// TIA Portal project "LearningFactory_4_0_24V_Task06_MultiProcessingMPO" (V16)

(* hardware
DEVICE "ET 200SP-Station_1"  ET 200SP-Station
   slot 0: "Baugruppenträger_0"  Rack  6ES5 710-8MAx1
   slot 1: "PLC"  CPU 1512SP-1 PN  6ES7 512-1DK01-0AB0  V2.8
      slot 32768: "PROFINET"  X1
   slot 2: "DO1+2"  DQ 16x24VDC/0.5A ST  6ES7 132-6BH01-0BA0  V0.0
      slot 1: "DO1+2"  DQ 16x24VDC/0.5A ST
   slot 3: "DO3+4"  DQ 16x24VDC/0.5A ST  6ES7 132-6BH01-0BA0  V0.0
      slot 1: "DO3+4"  DQ 16x24VDC/0.5A ST
   slot 4: "DO5+6"  DQ 16x24VDC/0.5A ST  6ES7 132-6BH01-0BA0  V0.0
      slot 1: "DO5+6"  DQ 16x24VDC/0.5A ST
   slot 5: "DO7-14"  DQ 4x24VDC/2A HS  6ES7 132-6BD20-0DA0  V2.0
      slot 1: "DO7-14"  DQ 4x24VDC/2A HS
   slot 6: "DO15-22"  DQ 4x24VDC/2A HS  6ES7 132-6BD20-0DA0  V2.0
      slot 1: "DO15-22"  DQ 4x24VDC/2A HS
   slot 7: "DO23-30"  DQ 4x24VDC/2A HS  6ES7 132-6BD20-0DA0  V2.0
      slot 1: "DO23-30"  DQ 4x24VDC/2A HS
   slot 8: "DI1+2"  DI 16x24VDC ST  6ES7 131-6BH01-0BA0  V0.0
      slot 1: "DI1+2"  DI 16x24VDC ST
   slot 9: "DI3+4"  DI 16x24VDC ST  6ES7 131-6BH01-0BA0  V0.0
      slot 1: "DI3+4"  DI 16x24VDC ST
   slot 10: "DI5"  DI 8x24VDC HS  6ES7 131-6BF00-0DA0  V1.0
      slot 1: "DI5"  DI 8x24VDC HS
   slot 11: "DI6"  DI 8x24VDC HS  6ES7 131-6BF00-0DA0  V1.0
      slot 1: "DI6"  DI 8x24VDC HS
   slot 12: "AI7-10"  AI 2xU ST  6ES7 134-6FB00-0BA1  V1.0
      slot 1: "AI7-10"  AI 2xU ST
   slot 13: "End"  Server module  6ES7 193-6PA00-0AA0  V1.1
      slot 1: "End"  Server module
   slot 127: "BA 2xRJ45"  BA 2xRJ45  6ES7 193-6AR00-0AA0  V0.0
      slot 32769: "Port_1"  6ES7 193-6AR00-0AA0
      slot 32770: "Port_2"  6ES7 193-6AR00-0AA0
*)

// ===== PLC "PLC"  CPU 1512SP-1 PN =====

VAR_GLOBAL   // PLC tag table "Start_Stop"
   "IX_START" AT %I4.4 : Bool;
   "IX_STOP" AT %I4.6 : Bool;
END_VAR

VAR_GLOBAL   // PLC tag table "MPO - Multi Processing Station with Oven"
   "IX_MPO_RefSwitchTurnTable_PosVac_I1" AT %I1.7 : Bool;
   "IX_MPO_RefSwitchTurnTable_PosBelt_I2" AT %I2.0 : Bool;
   "IX_MPO_LightBarrierEndOfConBelt_I3" AT %I2.1 : Bool;
   "IX_MPO_RefSwitchTurnTable_PosSaw_I4" AT %I2.2 : Bool;
   "IX_MPO_RefSwitchVac_PosTurnTable_I5" AT %I2.3 : Bool;
   "IX_MPO_RefSwitchOvenFeederInside_I6" AT %I2.4 : Bool;
   "IX_MPO_RefSwitchOvenFeederOutside_I7" AT %I2.5 : Bool;
   "IX_MPO_RefSwitchVac_PosOven_I8" AT %I2.6 : Bool;
   "IX_MPO_LightBarrierOven_I9" AT %I2.7 : Bool;
   "QX_MPO_M1_TurnTableClockwise_Q1" AT %Q3.0 : Bool;
   "QX_MPO_M1_TurnTableCounterclockwise_Q2" AT %Q3.1 : Bool;
   "QX_MPO_M2_ConveyorBeltForward_Q3" AT %Q3.2 : Bool;
   "QX_MPO_M3_Saw_Q4" AT %Q3.3 : Bool;
   "QX_MPO_M4_OvenFeederRetract_Q5" AT %Q3.4 : Bool;
   "QX_MPO_M4_OvenFeederExtend_Q6" AT %Q3.5 : Bool;
   "QX_MPO_M5_VacuumTowardsOven_Q7" AT %Q3.6 : Bool;
   "QX_MPO_M5_VacuumTowardsTurnTable_Q8" AT %Q3.7 : Bool;
   "QX_MPO_LightOven_Q9" AT %Q4.0 : Bool;
   "QX_MPO_Compressor_Q10" AT %Q4.1 : Bool;
   "QX_MPO_ValveVacuum_Q11" AT %Q4.2 : Bool;
   "QX_MPO_ValveLowering_Q12" AT %Q4.3 : Bool;
   "QX_MPO_ValveOvenDoor_Q13" AT %Q4.4 : Bool;
   "QX_MPO_ValveFeeder_Q14" AT %Q4.5 : Bool;
   "QW_MPO_PWM_TurnTable_M1" AT %QW23 : Int;
   "QW_MPO_PWM_Vacuum_M5" AT %QW25 : Int;
END_VAR

DATA_BLOCK "Task06_MultiProcessing_DB"   // DB4
{ S7_Optimized_Access := 'TRUE' }
VERSION : 0.1
// stored: InstanceOfName Task06_MultiProcessing
"Task06_MultiProcessing"
BEGIN
END_DATA_BLOCK

FUNCTION_BLOCK "Task06_MultiProcessing"   // FB4, SCL
{ S7_Optimized_Access := 'TRUE' }
VERSION : 0.1
   VAR_INPUT
      Start : Bool;
      Stop : Bool;
      RefSwitchTurnTable_PosVac : Bool;
      RefSwitchTurnTable_PosBelt : Bool;
      RefSwitchTurnTable_PosSaw : Bool;
      RefSwitchVac_PosTurnTable : Bool;
      RefSwitchVac_PosOven : Bool;
      RefSwitchOvenFeederInside : Bool;
      RefSwitchOvenFeederOutside : Bool;
      LightBarrierOven : Bool;
      LightBarrierEndOfConBelt : Bool;
   END_VAR
   VAR_OUTPUT
      M2_ConveyorBeltForward : Bool;
      M3_Saw : Bool;
      M4_OvenFeederRetract : Bool;
      M4_OvenFeederExtend : Bool;
      LightOven : Bool;
      PWM_TurnTable : Int;
      PWM_Vacuum : Int;
      Compressor : Bool;
   END_VAR
   VAR_IN_OUT
      M1_TurnTableClockwise : Bool;
      M1_TurnTableCounterclockwise : Bool;
      M5_VacuumTowardsOven : Bool;
      M5_VacuumTowardsTurnTable : Bool;
      ValveVacuum : Bool;
      ValveLowering : Bool;
      ValveOvenDoor : Bool;
      ValveFeeder : Bool;
   END_VAR
   VAR
      Step_number : Int;
      IEC_Timer_LoweringDown : TON_TIME;
      IEC_Timer_VacuumOn : TON_TIME;
      IEC_Timer_LoweringUp : TON_TIME;
      IEC_Timer_VacuumOff : TON_TIME;
      IEC_Timer_OvenClose : TON_TIME;
      IEC_Timer_OvenLight : TON_TIME;
      IEC_Timer_OvenOpen : TON_TIME;
      IEC_Timer_Saw : TON_TIME;
   END_VAR
BEGIN


   // Reset sequencer with pushbutton STOP 
   // Rücksetzen der Schrittkette  mit Taster STOP

   IF #Stop THEN
       #Step_number := 0;
   END_IF;

   // Start sequencer with pushbutton START
   // Starten der Schrittkette  mit Taster START

   CASE #Step_number OF
       0:  // Initial step 1 / Initialschritt 1
           #M2_ConveyorBeltForward := FALSE;           // Conveyor stop / Band stoppen  
           #M3_Saw := FALSE;                           // Saw off / Säge aus
           #M4_OvenFeederRetract := FALSE;             // Feeder oven retract stop / Ausschub Ofen einfahren stoppen
           #M4_OvenFeederExtend := FALSE;              // Feeder oven extend stop / Ausschub Ofen ausfahren stoppen 
           #LightOven := FALSE;                        // Light oven off / Licht im Ofen aus
           #M1_TurnTableClockwise := FALSE;            // Rotation clockwise stop / Rotation im Uhrzeigersinn stoppen
           #M1_TurnTableCounterclockwise := FALSE;     // Rotation counter clockwise stop / Rotation gegen den Uhrzeigersinn stoppen
           #M5_VacuumTowardsOven := FALSE;             // Linear axle towards oven stop / Linearachse zum Ofen stop 
           #M5_VacuumTowardsTurnTable := FALSE;        // Linear axle towards turn-table stop / Linearachse zum Drehtisch stop 
           #ValveVacuum := FALSE;                      // Vacuum gripper off / Vakuumgreifer aus
           #ValveLowering := FALSE;                    // Vacuum gripper up / Vakuumgreifer hoch
           #ValveOvenDoor := FALSE;                    // Door Oven close / Ofentüre schließen
           #ValveFeeder := FALSE;                      // Retract Zylinder feeder / Ausschubzylinder einfahren
           RESET_TIMER(#IEC_Timer_LoweringDown);       // Reset timer vacuum gripper down / Rücksetzen des Timers Vakuumgreifer abwärts
           RESET_TIMER(#IEC_Timer_VacuumOn);           // Reset timer vacuum on / Rücksetzen des Timers Vakuum ein
           RESET_TIMER(#IEC_Timer_LoweringUp);         // Reset timer vacuum gripper up / Rücksetzen des Timers Vakuumgreifer aufwärts
           RESET_TIMER(#IEC_Timer_VacuumOff);          // Reset timer vacuum off / Rücksetzen des Timers Vakuum aus
           RESET_TIMER(#IEC_Timer_OvenClose);          // Reset timer oven close / Rücksetzen des Timers Ofen schließen
           RESET_TIMER(#IEC_Timer_OvenLight);          // Reset timer light oven / Rücksetzen des Timers Licht im Ofen
           RESET_TIMER(#IEC_Timer_OvenOpen);           // Reset timer oven open / Rücksetzen des Timers Ofen öffnen
           RESET_TIMER(#IEC_Timer_Saw);                // Reset timer saw / Rücksetzen des Timers Säge

           IF #Start THEN
               #Step_number := #Step_number + 1;
           END_IF;

       1:  // Step 1 open oven; turn-table to position vacuum; linear axle towards turn-table
           // Schritt 1 Ofen öffnen; Drehtisch zu Position Vakuum; Linearachse zu Position Drehtisch
           #ValveOvenDoor := TRUE;                     // Door Oven open / Ofentüre öffnen
           #M1_TurnTableCounterclockwise := TRUE;      // Rotation counter clockwise / Rotation gegen den Uhrzeigersinn
           #M5_VacuumTowardsTurnTable := TRUE;         //Linear axle towards turn-table / Linearachse zum Drehtisch 

           IF #RefSwitchTurnTable_PosVac THEN
               #M1_TurnTableCounterclockwise := FALSE; // Rotation counter clockwise stop / Rotation gegen den Uhrzeigersinn stoppen
           END_IF;
           IF #RefSwitchVac_PosTurnTable THEN
               #M5_VacuumTowardsTurnTable := FALSE;    //Linear axle towards turn-table stop / Linearachse zum Drehtisch stop
           END_IF;

           IF #RefSwitchTurnTable_PosVac AND #RefSwitchVac_PosTurnTable THEN
               #Step_number := #Step_number + 1;
           END_IF;

       2:  // Step 2 vacuum gripper down / Schritt 2 Vakuumgreifer abwärts
           #ValveLowering := TRUE;                         // Vacuum gripper down / Vakuumgreifer abwärts
           #IEC_Timer_LoweringDown(IN := #ValveLowering,  // Start Timer vacuum gripper down / Timer starten Vakuumgreifer abwärts
                                PT := T#1s);

            IF #IEC_Timer_LoweringDown.Q THEN
                #Step_number := #Step_number + 1;
            END_IF;

        3:  // Step 3 vacuum on / Schritt 3 Vakuum ein
            #ValveVacuum := TRUE;                          // Vacuum on / Vakuum ein
            RESET_TIMER(#IEC_Timer_LoweringDown);          // Reset timer vacuum gripper down / Rücksetzen des Timers Vakuumgreifer abwärts
            #IEC_Timer_VacuumOn(IN := #ValveVacuum,        // Start Timer vacuum on / Timer starten Vakuum ein
                                    PT := T#1s);

            IF #IEC_Timer_VacuumOn.Q THEN
                #Step_number := #Step_number + 1;
            END_IF;

        4:  // Step 4 vacuum gripper up / Schritt 4 Vakuumgreifer aufwärts
            #ValveLowering := FALSE;                           // Vacuum gripper up / Vakuumgreifer aaufwärts
            RESET_TIMER(#IEC_Timer_VacuumOn);                  // Reset timer vacuum on / Rücksetzen des Timers Vakuum ein
            #IEC_Timer_LoweringUp(IN := NOT #ValveLowering,    // Start Timer vacuum gripper up / Timer starten Vakuumgreifer aufwärts
                                    PT := T#2s);

              IF #IEC_Timer_LoweringUp.Q THEN
                #Step_number := #Step_number + 1;
            END_IF;

        5:  // Step 5 extend feeder oven; linear axle towards oven
            // Schritt 5 Ausschub Ofen ausfahren; Linearachse zu Position Ofen
            #M4_OvenFeederExtend := TRUE;              // Feeder oven extend / Ausschub Ofen ausfahren 
            #M5_VacuumTowardsOven := TRUE;             // Linear axle towards oven / Linearachse zum Ofen
            RESET_TIMER(#IEC_Timer_LoweringUp);         // Reset timer vacuum gripper up / Rücksetzen des Timers Vakuumgreifer aufwärts

            IF #RefSwitchOvenFeederOutside THEN
                #M4_OvenFeederExtend := FALSE;         // Feeder oven extend stop / Ausschub Ofen ausfahren stoppen
            END_IF;
            IF #RefSwitchVac_PosOven THEN
                #M5_VacuumTowardsOven := FALSE;        //Linear axle towards oven stop / Linearachse zum Ofen stoppen
            END_IF;

            IF #RefSwitchOvenFeederOutside AND #RefSwitchVac_PosOven AND NOT #LightBarrierOven THEN
                #Step_number := #Step_number + 1;
            END_IF;

        6:  // Step 6 vacuum gripper down / Schritt 6 Vakuumgreifer abwärts
            #ValveLowering := TRUE;                         // Vacuum gripper down / Vakuumgreifer abwärts
            #IEC_Timer_LoweringDown(IN := #ValveLowering,  // Start Timer vacuum gripper down / Timer starten Vakuumgreifer abwärts
                                    PT := T#1s);

            IF #IEC_Timer_LoweringDown.Q THEN
                #Step_number := #Step_number + 1;
            END_IF;

        7:  // Step 7 vacuum off / Schritt 7 Vakuum aus
            #ValveVacuum := FALSE;                         // Vacuum off / Vakuum aus
            RESET_TIMER(#IEC_Timer_LoweringDown);          // Reset timer vacuum gripper down / Rücksetzen des Timers Vakuumgreifer abwärts
            #IEC_Timer_VacuumOff (IN := NOT #ValveVacuum,  // Start Timer vacuum off / Timer starten Vakuum off
                                PT := T#1s);

              IF #IEC_Timer_VacuumOff.Q THEN
                  #Step_number := #Step_number + 1;
              END_IF;

        8:  // Step 8 vacuum gripper up / Schritt 8 Vakuumgreifer aufwärts
            #ValveLowering := FALSE;                           // Vacuum gripper up / Vakuumgreifer aaufwärts
            RESET_TIMER(#IEC_Timer_VacuumOff);                 // Reset timer vacuum off / Rücksetzen des Timers Vakuum aus
            #IEC_Timer_LoweringUp(IN := NOT #ValveLowering,    // Start Timer vacuum gripper up / Timer starten Vakuumgreifer aufwärts
                                  PT := T#1s);

            IF #IEC_Timer_LoweringUp.Q THEN
                #Step_number := #Step_number + 1;
            END_IF;

        9:  // Step 9 retract feeder oven / Schritt 9 Ausschub Ofen einfahren
            #M4_OvenFeederRetract := TRUE;              // Feeder oven retract / Ausschub Ofen einfahren 
            RESET_TIMER(#IEC_Timer_LoweringUp);         // Reset Timer vacuum gripper up / Rücksetzen des Timers Vakuumgreifer aufwärts

            IF #RefSwitchOvenFeederInside THEN
                #Step_number := #Step_number + 1;
            END_IF;

       10:  // Step 10 close oven / Schritt 10 Ofen schließen
            #M4_OvenFeederRetract := FALSE;                    // Feeder oven retract off / Ausschub Ofen einfahren aus
            #ValveOvenDoor := FALSE;                           // Door Oven close / Ofentüre schließen
           #IEC_Timer_OvenClose(IN := NOT #ValveOvenDoor,     // Start Timer oven close / Starten des Timers Ofen schließen
                                  PT := T#1s);

             IF #IEC_Timer_OvenClose.Q THEN
                #Step_number := #Step_number + 1;
            END_IF;

        11:  // Step 11 light oven on / Schritt 11 Licht Ofen an
            #LightOven := TRUE;                        // Light oven on / Licht im Ofen an
            RESET_TIMER(#IEC_Timer_OvenClose);          // Reset timer oven close / Rücksetzen des Timers Ofen schließen
            #IEC_Timer_OvenLight(IN := #LightOven,     // Start Timer oven light / Starten des Timers Licht Ofen
                                 PT := T#5s);

            IF #IEC_Timer_OvenLight.Q THEN
                #Step_number := #Step_number + 1;
            END_IF;

        12:  // Step 12 open oven / Schritt 12 Ofen öffnen
            #LightOven := FALSE;                           // Light oven off / Licht im Ofen aus
            #ValveOvenDoor := TRUE;                        // Door Oven open / Ofentüre öffnen
            RESET_TIMER(#IEC_Timer_OvenLight);             // Reset timer light oven / Rücksetzen des Timers Licht im Ofen
            #IEC_Timer_OvenOpen(IN := #ValveOvenDoor,     // Start Timer oven open / Starten des Timers Ofen öffnen
                                 PT := T#1s);

             IF #IEC_Timer_OvenOpen.Q THEN
                #Step_number := #Step_number + 1;
            END_IF;

       13:  // Step 13 extend feeder oven / Schritt 13 Ausschub Ofen ausfahren
            #M4_OvenFeederExtend := TRUE;              // Feeder oven extend / Ausschub Ofen ausfahren 
            RESET_TIMER(#IEC_Timer_OvenOpen);           // Reset timer oven open / Rücksetzen des Timers Ofen öffnen

            IF #RefSwitchOvenFeederOutside THEN
                #Step_number := #Step_number + 1;
            END_IF;

       14:  // Step 14 vacuum gripper down; oven close / Schritt 14 Vakuumgreifer abwärts; Ofentüre schließen
            #ValveOvenDoor := FALSE;                        // Door Oven close / Ofentüre schließen
            #M4_OvenFeederExtend := FALSE;                  // Feeder oven extend off / Ausschub Ofen ausfahren aus
            #ValveLowering := TRUE;                         // Vacuum gripper down / Vakuumgreifer abwärts
            #IEC_Timer_LoweringDown(IN := #ValveLowering,  // Start Timer vacuum gripper down / Timer starten Vakuumgreifer abwärts
                                    PT := T#1s);

            IF #IEC_Timer_LoweringDown.Q THEN
                #Step_number := #Step_number + 1;
            END_IF;

       15:  // Step 15 vacuum on / Schritt 15 Vakuum ein
            #ValveVacuum := TRUE;                          // Vacuum on / Vakuum ein
            RESET_TIMER(#IEC_Timer_LoweringDown);          // Reset timer vacuum gripper down / Rücksetzen des Timers Vakuumgreifer abwärts
            #IEC_Timer_VacuumOn(IN := #ValveVacuum,        // Start Timer vacuum on / Timer starten Vakuum ein
                                PT := T#1s);

            IF #IEC_Timer_VacuumOn.Q THEN
                #Step_number := #Step_number + 1;
            END_IF;

        16:  // Step 16 vacuum gripper up / Schritt 16 Vakuumgreifer aufwärts
            #ValveLowering := FALSE;                           // Vacuum gripper up / Vakuumgreifer aaufwärts
            RESET_TIMER(#IEC_Timer_VacuumOn);                  // Reset timer vacuum on / Rücksetzen des Timers Vakuum ein
            #IEC_Timer_LoweringUp(IN := NOT #ValveLowering,    // Start Timer vacuum gripper up / Timer starten Vakuumgreifer aufwärts
                                  PT := T#2s);

            IF #IEC_Timer_LoweringUp.Q THEN
                #Step_number := #Step_number + 1;
            END_IF;

        17:  // Step 17 linear axle towards turn-table / Schritt 17 Linearachse zum Rundtisch
            #M5_VacuumTowardsTurnTable := TRUE;             // Linear axle towards turn-table / Linearachse zum Rundtisch
            RESET_TIMER(#IEC_Timer_LoweringUp);         // Reset timer vacuum gripper up / Rücksetzen des Timers Vakuumgreifer aufwärts

            IF #RefSwitchVac_PosTurnTable THEN
                #Step_number := #Step_number + 1;
            END_IF;

        18:  // Step 18 vacuum gripper down / Schritt 18 Vakuumgreifer abwärts
            #M5_VacuumTowardsTurnTable := FALSE;             // Linear axle towards turn-table off / Linearachse zum Rundtisch aus
            #ValveLowering := TRUE;                         // Vacuum gripper down / Vakuumgreifer abwärts
            #IEC_Timer_LoweringDown(IN := #ValveLowering,  // Start Timer vacuum gripper down / Timer starten Vakuumgreifer abwärts
                                    PT := T#1s);

            IF #IEC_Timer_LoweringDown.Q THEN
                #Step_number := #Step_number + 1;
            END_IF;

       19:  // Step 7 vacuum off / Schritt 19 Vakuum aus
            #ValveVacuum := FALSE;                         // Vacuum off / Vakuum aus
            RESET_TIMER(#IEC_Timer_LoweringDown);          // Reset timer vacuum gripper down / Rücksetzen des Timers Vakuumgreifer abwärts
            #IEC_Timer_VacuumOff(IN := NOT #ValveVacuum,  // Start Timer vacuum off / Timer starten Vakuum off
                                 PT := T#1s);

            IF #IEC_Timer_VacuumOff.Q THEN
                #Step_number := #Step_number + 1;
            END_IF;

       20:  // Step 20 vacuum gripper up / Schritt 20 Vakuumgreifer aufwärts
            #ValveLowering := FALSE;                           // Vacuum gripper up / Vakuumgreifer aaufwärts
            RESET_TIMER(#IEC_Timer_VacuumOff);                 // Reset timer vacuum off / Rücksetzen des Timers Vakuum aus
            #IEC_Timer_LoweringUp(IN := NOT #ValveLowering,    // Start Timer vacuum gripper up / Timer starten Vakuumgreifer aufwärts
                                  PT := T#1s);

            IF #IEC_Timer_LoweringUp.Q THEN
                #Step_number := #Step_number + 1;
            END_IF;

       21:  // Step 21 rotation clockwise to position saw / Schritt 21 Rotation im Uhrzeigersinn zur Position Säge
           #M1_TurnTableClockwise := TRUE;            // Rotation clockwise / Rotation im Uhrzeigersinn
            RESET_TIMER(#IEC_Timer_LoweringUp);         // Reset Timer vacuum gripper up / Rücksetzen des Timers Vakuumgreifer aufwärts

            IF #RefSwitchTurnTable_PosSaw THEN
                #Step_number := #Step_number + 1;
            END_IF;

       22:  // Step 22 saw on 5 seconds / Schritt 22 Säge ein 5 Sekunden
            #M1_TurnTableClockwise := FALSE;            // Rotation clockwise stop/ Rotation im Uhrzeigersinn stoppen
            #M3_Saw := TRUE;                           // Saw on / Säge ein
            #IEC_Timer_Saw(IN := #M3_Saw,    // Start Timer saw on / Timer starten Säge ein
                                  PT := T#5s);

            IF #IEC_Timer_Saw.Q THEN
                #Step_number := #Step_number + 1;
            END_IF;

       23:  // Step 23 rotation clockwise to position conveyorbelt/ Schritt 23 Rotation im Uhrzeigersinn zum Förderband
            #M3_Saw := FALSE;                           // Saw off / Säge aus
            #M1_TurnTableClockwise := TRUE;            // Rotation clockwise / Rotation im Uhrzeigersinn
            RESET_TIMER(#IEC_Timer_Saw);                // Reset timer saw / Rücksetzen des Timers Säge

            IF #RefSwitchTurnTable_PosBelt THEN
               #Step_number := #Step_number + 1;
           END_IF;

       24:  // Step 24 extend feeder; start conveyorbelt/ Schritt 24 Ausschubzylinder ausfahren; Band starten
               #M1_TurnTableClockwise := FALSE;            // Rotation clockwise off / Rotation im Uhrzeigersinn aus
               #ValveFeeder := TRUE;                      // Extend Zylinder feeder / Ausschubzylinder ausfahren
               #M2_ConveyorBeltForward := TRUE;           // Conveyorbelt start / Band starten 

               IF #LightBarrierEndOfConBelt THEN
                   #Step_number := #Step_number + 1;
               END_IF;

       25:  // Step 25 end of sequencer / Schritt 24 Schrittkettenende
               #ValveFeeder := FALSE;                          // Retract Zylinder feeder / Ausschubzylinder einfahren
               #M2_ConveyorBeltForward := FALSE;              // Conveyorbelt stop / Band stoppen

               IF NOT #ValveFeeder AND NOT #M2_ConveyorBeltForward THEN
                   #Step_number :=0;
               END_IF;

           ELSE  // Statement section ELSE
           ;
   END_CASE;


   //Permanent Instructions

   //Pulse width modulation control for turn-table 
   //Pulsweitenmodulation für Drehtisch
   IF #M1_TurnTableClockwise OR #M1_TurnTableCounterclockwise
   THEN
       #PWM_TurnTable := 500;
   ELSE
       #PWM_TurnTable := 0;
   END_IF;

   //Pulse width modulation control for linear axle vacuum gripper
   //Pulsweitenmodulation für Linearachse Vakuumgreifer
   IF #M5_VacuumTowardsOven OR #M5_VacuumTowardsTurnTable
   THEN
       #PWM_Vacuum := 700;
   ELSE
       #PWM_Vacuum := 0;
   END_IF;

   // Compressor on / Kompressor ein
   IF #ValveVacuum OR #ValveLowering
       OR #ValveOvenDoor OR #ValveFeeder
   THEN
       #Compressor := TRUE;
   ELSE
       #Compressor := FALSE;
   END_IF;
END_FUNCTION_BLOCK

ORGANIZATION_BLOCK "Main"   // OB1, SCL, ProgramCycle
TITLE = "Main Program Sweep (Cycle)"
{ S7_Optimized_Access := 'TRUE' }
VERSION : 0.1
   VAR_INPUT
      Initial_Call : Bool;   // Initial call of this OB
      Remanence : Bool;   // =True, if remanent data are available
   END_VAR
BEGIN


   // Call subroutine VacuumGripper
   // Aufruf Unterprogramm VacuumGripper


   "Task06_MultiProcessing_DB"(Start:="IX_START",
                               Stop:= NOT "IX_STOP",
                               RefSwitchTurnTable_PosVac:="IX_MPO_RefSwitchTurnTable_PosVac_I1",
                               RefSwitchTurnTable_PosBelt:="IX_MPO_RefSwitchTurnTable_PosBelt_I2",
                               RefSwitchTurnTable_PosSaw:="IX_MPO_RefSwitchTurnTable_PosSaw_I4",
                               RefSwitchVac_PosTurnTable:="IX_MPO_RefSwitchVac_PosTurnTable_I5",
                               RefSwitchVac_PosOven:="IX_MPO_RefSwitchVac_PosOven_I8",
                               RefSwitchOvenFeederInside:="IX_MPO_RefSwitchOvenFeederInside_I6",
                               RefSwitchOvenFeederOutside:="IX_MPO_RefSwitchOvenFeederOutside_I7",
                               LightBarrierOven:= NOT "IX_MPO_LightBarrierOven_I9",
                               LightBarrierEndOfConBelt:= NOT "IX_MPO_LightBarrierEndOfConBelt_I3",
                               M1_TurnTableClockwise:="QX_MPO_M1_TurnTableClockwise_Q1",
                               M1_TurnTableCounterclockwise:="QX_MPO_M1_TurnTableCounterclockwise_Q2",
                               PWM_TurnTable=>"QW_MPO_PWM_TurnTable_M1",
                               M2_ConveyorBeltForward=>"QX_MPO_M2_ConveyorBeltForward_Q3",
                               M3_Saw=>"QX_MPO_M3_Saw_Q4",
                               M4_OvenFeederRetract=>"QX_MPO_M4_OvenFeederRetract_Q5",
                               M4_OvenFeederExtend=>"QX_MPO_M4_OvenFeederExtend_Q6",
                               M5_VacuumTowardsOven:="QX_MPO_M5_VacuumTowardsOven_Q7",
                               M5_VacuumTowardsTurnTable:="QX_MPO_M5_VacuumTowardsTurnTable_Q8",
                               PWM_Vacuum=>"QW_MPO_PWM_Vacuum_M5",
                               LightOven=>"QX_MPO_LightOven_Q9",
                               ValveVacuum:="QX_MPO_ValveVacuum_Q11",
                               ValveLowering:="QX_MPO_ValveLowering_Q12",
                               ValveOvenDoor:="QX_MPO_ValveOvenDoor_Q13",
                               ValveFeeder:="QX_MPO_ValveFeeder_Q14",
                               Compressor=>"QX_MPO_Compressor_Q10");
END_ORGANIZATION_BLOCK